(* IEC 61131-3 sources: UnioviWaterTanks/ME_TANK_TP, 4 files *)

(* ---- DT_Tank.st ---- *)
TYPE DT_TANK
STRUCT

Identifier : real; (**)
(*Entradas y salidas fisicas del tanque*)

// Temp_TP := REAL; // Temperatura instantanea del bloque
Nivel : REAL; // Nivel instantaneo del bloque

Max : BOOL; // Sensor de nivel maximo; Normalmente abierto
Min :BOOL; // Sensor de nivel minimo; Normalmente cerradp

V1 : BOOL; // Accionamiento sobre la valvula V1, conecta DS -> TP
V2 : BOOL; // Accionamiento sobre la valvula V2, conecta TP -> DI
V3 : bool; // Accionamiento sobre la valvula V3, conecta TP -> TP // TP -> DS
V5 : BOOL; // Accionamiento sobre la valvula ternaria V3

(*Parametros de funcionamiento*)

(*Parametros de supervisión*)

(*Estados de funcionamiento*)
Llenado : bool;
Vaciado : bool;
Vacio : bool;
LLeno : bool;

END_STRUCT
END_TYPE

(* ---- FB_MoveAllFluid.st ---- *)
FUNCTION_BLOCK FB_MoveAllFluid
(*BLOQUE FUNCIONAL DEL TANQUE: MOVE ALL FLUID*)
(*=================================================================================*)

(*DESCRIPCIÓN: Bloque funcional que a partir de dos tanques se encarga de comprobar
que se cumplen las restricciones locales de funcionamiento, es decir,
que el tanque que cede o GuestTank tenga fluido y que el tanque que recive o
HostTank no este al maximo de su capacidad.
Ademas a partir del conocimiento del esquema de conexiones del sistema
implementamos un codigo encargado de asignar a cada tanque las conexiones
con las valvulas correspondientes para el movimiento de fluido adecuado
Para realizar esto, se ha codificado el tanque con un numero identificador
que podemos encontrar en la estructura llamada DataType. La codificacion es del 0
al n-1 tanques siendo los numeros mas bajos los que se encuentran en la
parte superior del sistema. En este caso en concreto: DS -> 0,TP -> 1, DS ->2*)

VAR_INPUT
Enable : BOOL; (*Condicion de funcionamiento en el nivel mas exterior del bloque*)

Iniciar : bool; (*Condicion de inicio del proceso*)

TDone : Real; (*Tiempo de establecimiento de la señal de finalizacion*)
END_VAR

VAR_IN_OUT
GuestTank : DT_Tank; (*Data Type del tanque que cede fluido,*)
HostTank : DT_Tank; (*Data Type del tanque que recive el fluido*)
END_VAR

VAR_OUTPUT
MSG : STRING; (*Muestra mensajes de informacion relevante para el sistema*)
OUT_Comand_V1 : bool; (*Gobierna la valvula V1 en los estados de ON/OFF*)
OUT_Comand_V2 : bool; (*Gobierna la valvula V2 en los estados de ON/OFF*)
OUT_Comand_V3 : bool; (*Gobierna la valvula V3 en los estados de ON/OFF*)
OUT_Comand_V4 : bool; (*Gobierna la valvula V4 en los estados de ON/OFF*)
OUT_Comand_V5_1 : bool; (*Gobierna la valvula V5.1 en los estados de ON/OFF*)
OUT_Comand_V5_2 : bool; (*Gobierna la valvula V5.2 en los estados de ON/OFF*)
OUT_Power_B2 : Real;(*Fija la potencia aplicada al actuador*)

Done : bool; (*Señal que indica cuando ha finalizado la accion*)
END_VAR

VAR
//Finalizar : BOOL; (*Condicion de finalizacion del proceso*)
//Permiso : BOOL; (*Condicion de funcionamiento local*)
EmptyAllTank : FB_TankBasic;
END_VAR

(*CODIGO DE FUNCIONAMIENTO*)
(*=================================================================================*)
EmptyAllTank (Enable := Enable,
			  Permiso := GuestTank.Maximo AND NOT HostTank.Maximo,
              Iniciar := Iniciar,
			  Finalizar := NOT GuestTank.Minimo OR HostTank.Minimo,
              TDone := TDone);

(*Independientemente del Deposito que se este llenando, señalamos
el cambio en los estados de los dos depositos*)
GuestTank.State := 'Vaciandose';
HostTank.State := 'Llenandose';

(*GESTION DE CONEXION DE LAS VALVULAS*)
(******************************************************************************)

(*Conexiones del DEPOSITO SUPERIOR*)

IF GuestTank.Identifier = 0 THEN
  IF HostTank.Identifier = 1 THEN
     (*Conexion Deposito Superior con Tanque Principal*)
      MSG := '(DS -> TP) Fluyendo';
      OUT_Comand_V1 := EmptyAllTank.OUT_Comand;
      OUT_Comand_V2 := FALSE;
      OUT_Comand_V3 := FALSE;
      OUT_Comand_V4 := FALSE;
      OUT_Comand_V5_1 := FALSE;
      OUT_Comand_V5_2 := FALSE;
      OUT_Power_B2 := 0.0; // En este caso la Bomba no funciona
	END_IF;
	IF HostTank.Identifier = 2 THEN
     (*Conexion Deposito Superior con Deposito Inferior 'pasando por TP'*)
    (*Como pasa por TP podria ser necesario tener en cuenta el nivel del tanque
     pero si lo asimilamos a una tuberia, ya que le llega fluido y sale de el con
     el mismo caudal el nivel del tanque queda invariable y es como si existiese
     una tuberia que conecta los dos depositos*)
      MSG := '(DS -> TP -> DI) Fluyendo';
      OUT_Comand_V1 := EmptyAllTank.OUT_Comand;
      OUT_Comand_V2 := EmptyAllTank.OUT_Comand;
      OUT_Comand_V3 := FALSE;
      OUT_Comand_V4 := FALSE;
      OUT_Comand_V5_1 := FALSE;
      OUT_Comand_V5_2 := FALSE;
      OUT_Power_B2 := 0.0; // En este caso la Bomba no funciona
	END_IF;

END_IF;

(*Conexiones del TANQUE PRINCIPAL*)

IF GuestTank.Identifier = 1 THEN
  IF HostTank.Identifier = 0 THEN
    (*Conexion Tanque Principal con Deposito Superior*)
    MSG := '(TP -> DS) Fluyendo';
    OUT_Comand_V1 := FALSE;
    OUT_Comand_V2 := FALSE;
    OUT_Comand_V3 := EmptyAllTank.OUT_Comand;
    OUT_Comand_V4 := FALSE;
    OUT_Comand_V5_1 := FALSE;
    OUT_Comand_V5_2 := EmptyAllTank.OUT_Comand;
    OUT_Power_B2 := HostTank.Power; // Fijamos la potencia de la bomba segun HostTank
	END_IF;
	IF HostTank.Identifier = 2 THEN
    (*Conexion Tanque Principal con Deposito Inferior*)
    MSG := '(TP -> DI) Fluyendo';
    OUT_Comand_V1 := FALSE;
    OUT_Comand_V2 := EmptyAllTank.OUT_Comand;
    OUT_Comand_V3 := FALSE;
    OUT_Comand_V4 := FALSE;
    OUT_Comand_V5_1 := FALSE;
    OUT_Comand_V5_2 := FALSE;
    OUT_Power_B2 := 0.0; // En este caso la Bomba no funciona
	END_IF;
END_IF;

(*Conexiones del DEPOSITO INFERIOR*)

IF GuestTank.Identifier = 2 THEN
  IF HostTank.Identifier = 0 THEN
    (*Conexion Deposito Inferior con Deposito Superior*)
    MSG := '(DI -> DS) Fluyendo';
    OUT_Comand_V1 := FALSE;
    OUT_Comand_V2 := FALSE;
    OUT_Comand_V3 := FALSE;
    OUT_Comand_V4 := EmptyAllTank.OUT_Comand;
    OUT_Comand_V5_1 := FALSE;
    OUT_Comand_V5_2 := EmptyAllTank.OUT_Comand;
    OUT_Power_B2 := HostTank.Power; // Fijamos la potencia de la bomba segun HostTank
	END_IF
	IF HostTank.Identifier = 1 THEN
    (*Conexion Deposito Inferior con Tanque Principal*)
    MSG := '(DI -> TP) Fluyendo';
    OUT_Comand_V1 := FALSE;
    OUT_Comand_V2 := FALSE;
    OUT_Comand_V3 := FALSE;
    OUT_Comand_V4 := EmptyAllTank.OUT_Comand;
    OUT_Comand_V5_1 := EmptyAllTank.OUT_Comand;
    OUT_Comand_V5_2 := FALSE;
    OUT_Power_B2 := HostTank.Power; // Fijamos la potencia de la bomba segun HostTank
	END_IF;
END_IF;

(* ---- FB_EmptyAll.st ---- *)
(*BLOQUE FUNCIONAL DEL TANQUE: EMPTY ALL*)
(*=================================================================================*)

(*DESCRIPCIÓN: Bloque funcional que vacia el tanque principal, *)
VAR_INPUT
Enable : BOOL; (*Condicion de funcionamiento en el nivel mas exterior del bloque*)
Permiso : BOOL; (*Condicion de funcionamiento local*)
Iniciar : bool; (*Condicion de inicio del proceso*)
Finalizar : bool; (*Condicion de finalizacion del proceso*)
TDone : Real; (*Tiempo de establecimiento de la señal de finalizacion*)
END_VAR

var_IN_OUT
GuestTank : DT_Tank; (*Data Type del tanque que cede fluido,*)
HostTank : DT_Tank; (*Data Type del tanque que recive el fluido*)
END_VAR

VAR_OUTPUT
MSG : STRING; (*Muestra mensajes de informacion relevante para el sistema*)
OUT_Power : real; (*Fija la potencia aplicada al actuador*)
OUT_Comand : Bool; (*Gobierna el actuador en los estados de ON/OFF*)
Done : bool; (*Señal que indica cuando ha finalizado la accion*)
END_VAR

var
EmptyAllTank : FB_TankBasic;
END_VAR

(*CODIGO DE FUNCIONAMIENTO*)

EmptyAllTank (Enable := Enable,
              Permiso := GuestTank.Max and not HostTank.Max,
              )

(* ---- FB_TankBasic.st ---- *)
(**)

(*BLOQUE FUNCIONAL PARA EL DESARROLLO DE ACCIONES DEL MODULO DE EQUIPAMIENTO TANQUE*)
(*=================================================================================*)

(*DEFINICIÓN DE LAS VARIABLES*)
VAR_INPUT
Enable : BOOL; (*Condicion de funcionamiento en el nivel mas exterior del bloque*)
Permiso : BOOL; (*Condicion de funcionamiento local*)
Iniciar : bool; (*Condicion de inicio del proceso*)
Finalizar : bool; (*Condicion de finalizacion del proceso*)
TDone : Real; (*Tiempo de establecimiento de la señal de finalizacion)
//DI_DS := Bool; (*Seleccion del deposito de Origen/Destino*)
END_VAR

//var_IN_OUT
//Estado := int; (*Indica el estado anterior del modulo de equipamiento*)
//END_VAR

VAR_OUTPUT
MSG : STRING; (*Muestra mensajes de informacion relevante para el sistema*)
OUT_Power : real; (*Fija la potencia aplicada al actuador*)
OUT_Comand : Bool; (*Gobierna el actuador en los estados de ON/OFF*)
Done : bool; (*Señal que indica cuando ha finalizado la accion*)
END_VAR

var
RS_ON_OFF : RS; (*Bloque RS*)
F_EdgeDetection : F_TRIG; (*Falling Edge Detection*)
Fin : TP (*Pulse Timer, donde IN es la activacion y PT la duracion del pulso*)
END_VAR

(*CODIGO DE FUNCIONAMIENTO*)

  IF Enable THEN

    MSG := '    '; (*Mensaje*)
    RS_ON_OFF (SET := Iniciar AND Permiso, RESET := Finalizar)

    Actuador := RS_Act.Q1 AND Permiso;

    if Actuador THEN

      MSG:= 'Actuador activado'; // Indicamos que el bloque funciona
      OUT_Comand := True; (*Encendemos el actuador*)
      OUT_Power := SP_Power ; // Fijamos la potencia de salida

    else
        OUT_Comand := False; (*Actuador apagado*)
        OUT_Power := 0.0; (*Potencia de salida = 0*)

    END_IF

    F_EdgeDetection (CLK:=Actuador);
    (*Generamos un flanco cuando Actuador pasa de 0->1 que nos sirve para
    activar un temporizador de tiempo 'TDone'*)

    Fin (IN:= F_EdgeDetection.Q,PT:=TO_TIME(TDone));
    (*El flanco activa el temporizador 'Fin'*)

    Done := Fin.Q; (*Durante TDone señalaremos con la señal Done que la
      accion ha terminado*)

    if Done THEN
      MSG := 'Finalizado';
    END_IF

    END_IF

  END_IF
